PROGRAM TSCS_Bridge_Inputs	
(* Inputs from TSCS PLC to TDU PLC*)
VAR
	// Function Blocks
	BYTE_TO_BITS_10: OSCAT_BYTE_TO_BITS; // Interface for TSCS Byte 0 - Boolean inputs
	BYTE_TO_BITS_11: OSCAT_BYTE_TO_BITS; // Interface for TSCS Byte 1 - Boolean inputs
	BYTE_TO_BITS_12: OSCAT_BYTE_TO_BITS; // Interface for TSCS Byte 2 - Boolean inputs
	BYTE_TO_BITS_13: OSCAT_BYTE_TO_BITS; // Interface for TSCS Byte 3 - Boolean inputs
	BYTE_TO_BITS_14: OSCAT_BYTE_TO_BITS; // Interface for TSCS Byte 4 - Boolean inputs
	BYTE_TO_BITS_20: OSCAT_BYTE_TO_BITS; // Interface for TMS Byte 0 - Boolean inputs
	BYTE_TO_BITS_21: OSCAT_BYTE_TO_BITS; // Interface for TMS Byte 1 - Boolean inputs
	BYTE_TO_BITS_22: OSCAT_BYTE_TO_BITS; // Interface for TMS Byte 2 - Boolean inputs
	BYTE_TO_BITS_23: OSCAT_BYTE_TO_BITS; // Interface for TMS Byte 3 - Boolean inputs
	BYTE_TO_BITS_24: OSCAT_BYTE_TO_BITS; // Interface for TMS Byte 4 - Boolean inputs
	fb_Bridge_Integer_Inputs_0 : FB_Bridge_Inputs_Integer; // Interface for TSCS Integers
	fb_Bridge_Integer_Inputs_1 : FB_Bridge_Inputs_Integer; // Interface for TMS Integers
	fb_Bridge_Real_Inputs_0 : FB_Bridge_Inputs_Real; // Interface for TSCS real signals
	fb_Bridge_Real_Inputs_1 : FB_Bridge_Inputs_Real; // Interface for TMS real signals
	
	// Test Signal
	TDU_TestSignal_RB : REAL;	// Diagnostic signal readback (TDU -> TSCS ->TDU)
		
	// TSCS signals (as example)
	Lube_MainBearing_Act : BOOL; 		// Main bearing lubrication active
	TSCS_State : INT; 					// Target System Operation Mode [0=Off, 1=Normal Operation, 2=Maintenance]
	Lube_MainBearing_FlowRate : REAL; 	// Main bearing lubrication flow rate [mL/min]
END_VAR

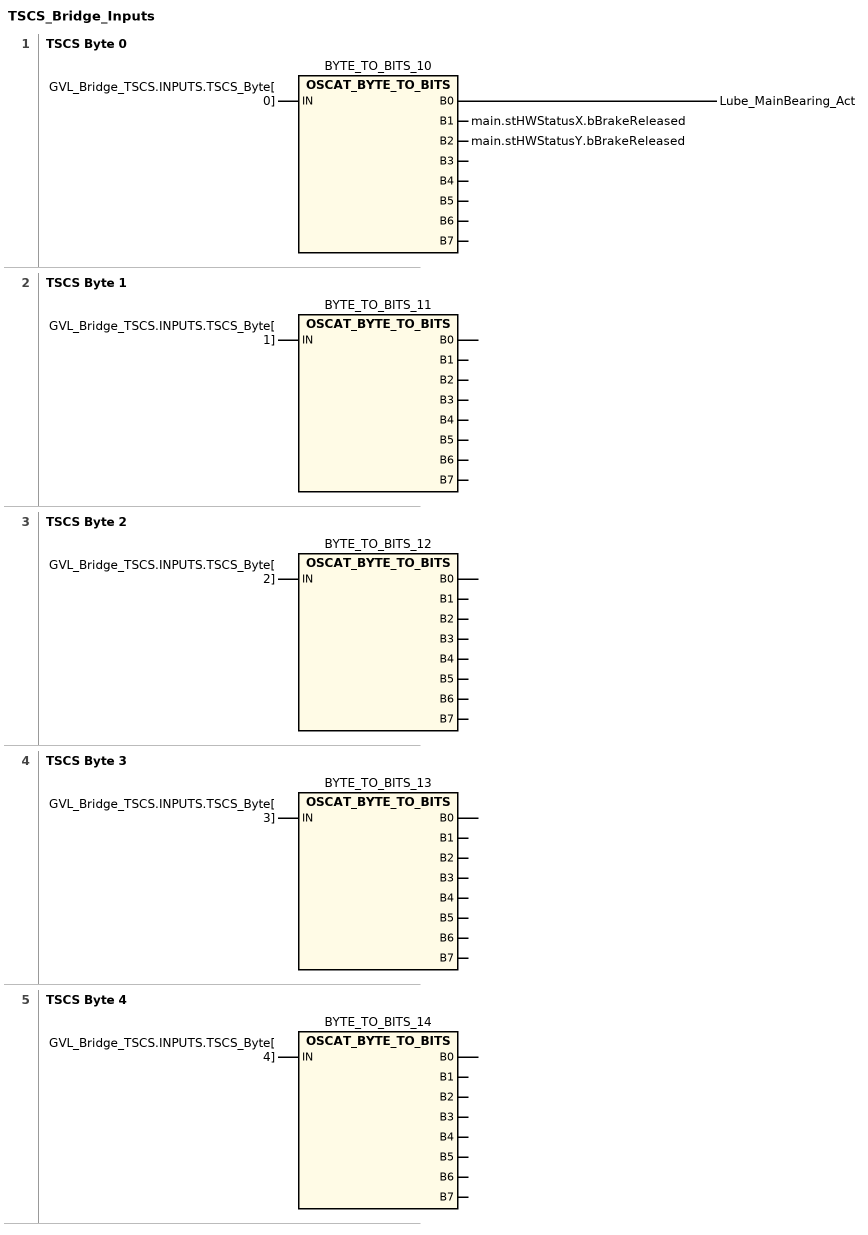
// NETWORK 1: TSCS Byte 0
BYTE_TO_BITS_10(
    IN := GVL_Bridge_TSCS.INPUTS.TSCS_Byte[0],
    B1 => main.stHWStatusX.bBrakeReleased,
    B2 => main.stHWStatusY.bBrakeReleased); // OSCAT_BYTE_TO_BITS
Lube_MainBearing_Act := BYTE_TO_BITS_10.B0;

// NETWORK 2: TSCS Byte 1
BYTE_TO_BITS_11(IN := GVL_Bridge_TSCS.INPUTS.TSCS_Byte[1]); // OSCAT_BYTE_TO_BITS

// NETWORK 3: TSCS Byte 2
BYTE_TO_BITS_12(IN := GVL_Bridge_TSCS.INPUTS.TSCS_Byte[2]); // OSCAT_BYTE_TO_BITS

// NETWORK 4: TSCS Byte 3
BYTE_TO_BITS_13(IN := GVL_Bridge_TSCS.INPUTS.TSCS_Byte[3]); // OSCAT_BYTE_TO_BITS

// NETWORK 5: TSCS Byte 4
BYTE_TO_BITS_14(IN := GVL_Bridge_TSCS.INPUTS.TSCS_Byte[4]); // OSCAT_BYTE_TO_BITS

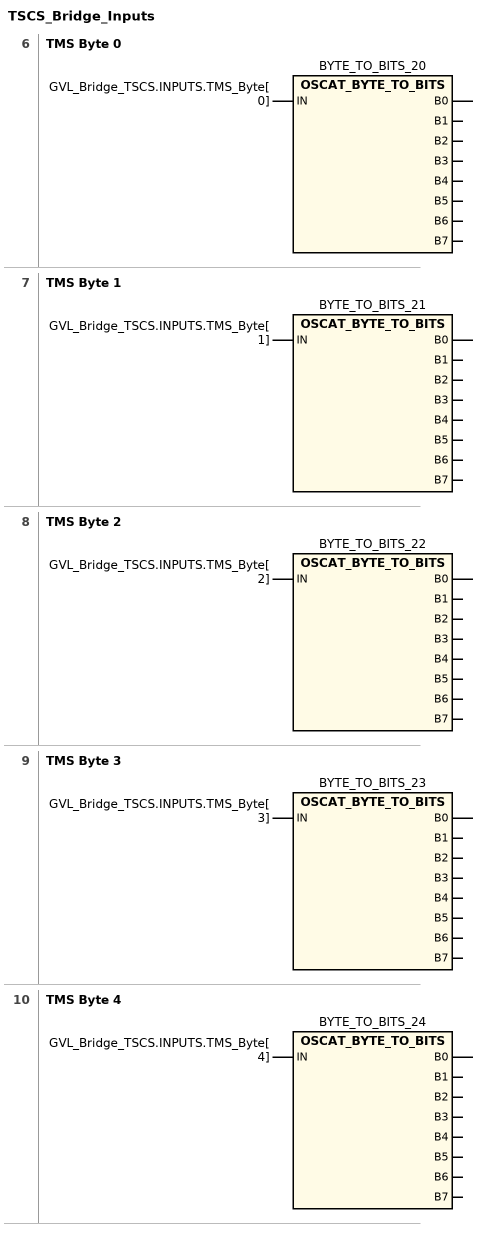
// NETWORK 6: TMS Byte 0
BYTE_TO_BITS_20(IN := GVL_Bridge_TSCS.INPUTS.TMS_Byte[0]); // OSCAT_BYTE_TO_BITS

// NETWORK 7: TMS Byte 1
BYTE_TO_BITS_21(IN := GVL_Bridge_TSCS.INPUTS.TMS_Byte[1]); // OSCAT_BYTE_TO_BITS

// NETWORK 8: TMS Byte 2
BYTE_TO_BITS_22(IN := GVL_Bridge_TSCS.INPUTS.TMS_Byte[2]); // OSCAT_BYTE_TO_BITS

// NETWORK 9: TMS Byte 3
BYTE_TO_BITS_23(IN := GVL_Bridge_TSCS.INPUTS.TMS_Byte[3]); // OSCAT_BYTE_TO_BITS

// NETWORK 10: TMS Byte 4
BYTE_TO_BITS_24(IN := GVL_Bridge_TSCS.INPUTS.TMS_Byte[4]); // OSCAT_BYTE_TO_BITS

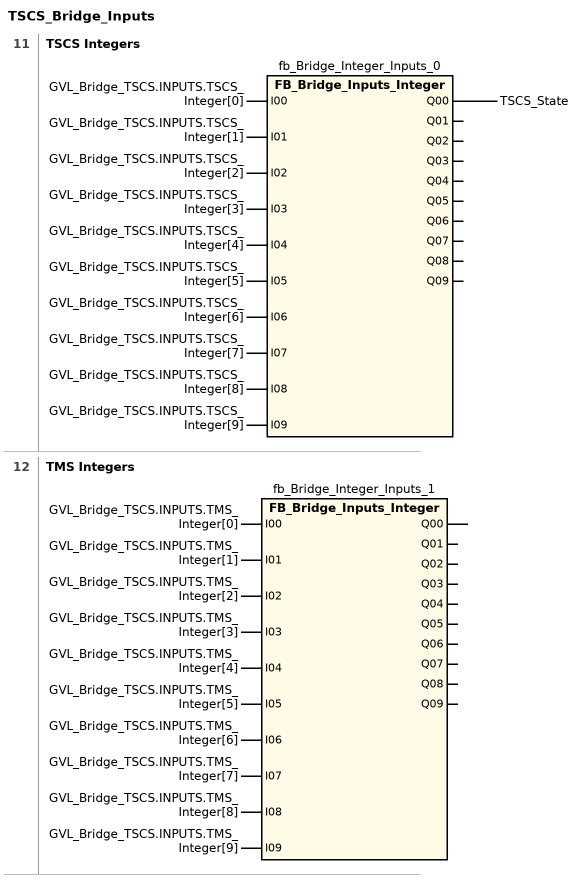
// NETWORK 11: TSCS Integers
fb_Bridge_Integer_Inputs_0(
    I00 := GVL_Bridge_TSCS.INPUTS.TSCS_Integer[0],
    I01 := GVL_Bridge_TSCS.INPUTS.TSCS_Integer[1],
    I02 := GVL_Bridge_TSCS.INPUTS.TSCS_Integer[2],
    I03 := GVL_Bridge_TSCS.INPUTS.TSCS_Integer[3],
    I04 := GVL_Bridge_TSCS.INPUTS.TSCS_Integer[4],
    I05 := GVL_Bridge_TSCS.INPUTS.TSCS_Integer[5],
    I06 := GVL_Bridge_TSCS.INPUTS.TSCS_Integer[6],
    I07 := GVL_Bridge_TSCS.INPUTS.TSCS_Integer[7],
    I08 := GVL_Bridge_TSCS.INPUTS.TSCS_Integer[8],
    I09 := GVL_Bridge_TSCS.INPUTS.TSCS_Integer[9]); // FB_Bridge_Inputs_Integer
TSCS_State := fb_Bridge_Integer_Inputs_0.Q00;

// NETWORK 12: TMS Integers
fb_Bridge_Integer_Inputs_1(
    I00 := GVL_Bridge_TSCS.INPUTS.TMS_Integer[0],
    I01 := GVL_Bridge_TSCS.INPUTS.TMS_Integer[1],
    I02 := GVL_Bridge_TSCS.INPUTS.TMS_Integer[2],
    I03 := GVL_Bridge_TSCS.INPUTS.TMS_Integer[3],
    I04 := GVL_Bridge_TSCS.INPUTS.TMS_Integer[4],
    I05 := GVL_Bridge_TSCS.INPUTS.TMS_Integer[5],
    I06 := GVL_Bridge_TSCS.INPUTS.TMS_Integer[6],
    I07 := GVL_Bridge_TSCS.INPUTS.TMS_Integer[7],
    I08 := GVL_Bridge_TSCS.INPUTS.TMS_Integer[8],
    I09 := GVL_Bridge_TSCS.INPUTS.TMS_Integer[9]); // FB_Bridge_Inputs_Integer

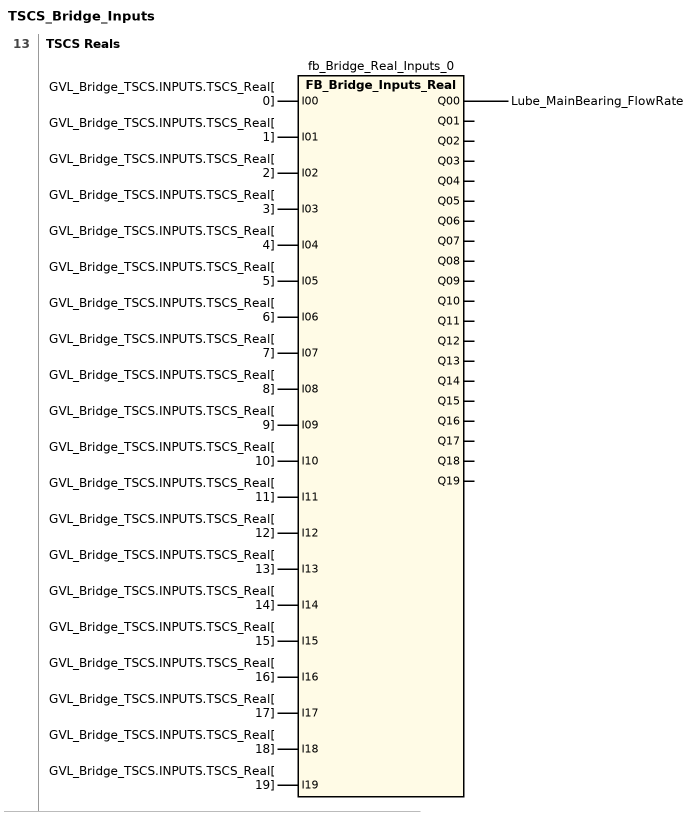
// NETWORK 13: TSCS Reals
fb_Bridge_Real_Inputs_0(
    I00 := GVL_Bridge_TSCS.INPUTS.TSCS_Real[0],
    I01 := GVL_Bridge_TSCS.INPUTS.TSCS_Real[1],
    I02 := GVL_Bridge_TSCS.INPUTS.TSCS_Real[2],
    I03 := GVL_Bridge_TSCS.INPUTS.TSCS_Real[3],
    I04 := GVL_Bridge_TSCS.INPUTS.TSCS_Real[4],
    I05 := GVL_Bridge_TSCS.INPUTS.TSCS_Real[5],
    I06 := GVL_Bridge_TSCS.INPUTS.TSCS_Real[6],
    I07 := GVL_Bridge_TSCS.INPUTS.TSCS_Real[7],
    I08 := GVL_Bridge_TSCS.INPUTS.TSCS_Real[8],
    I09 := GVL_Bridge_TSCS.INPUTS.TSCS_Real[9],
    I10 := GVL_Bridge_TSCS.INPUTS.TSCS_Real[10],
    I11 := GVL_Bridge_TSCS.INPUTS.TSCS_Real[11],
    I12 := GVL_Bridge_TSCS.INPUTS.TSCS_Real[12],
    I13 := GVL_Bridge_TSCS.INPUTS.TSCS_Real[13],
    I14 := GVL_Bridge_TSCS.INPUTS.TSCS_Real[14],
    I15 := GVL_Bridge_TSCS.INPUTS.TSCS_Real[15],
    I16 := GVL_Bridge_TSCS.INPUTS.TSCS_Real[16],
    I17 := GVL_Bridge_TSCS.INPUTS.TSCS_Real[17],
    I18 := GVL_Bridge_TSCS.INPUTS.TSCS_Real[18],
    I19 := GVL_Bridge_TSCS.INPUTS.TSCS_Real[19]); // FB_Bridge_Inputs_Real
Lube_MainBearing_FlowRate := fb_Bridge_Real_Inputs_0.Q00;

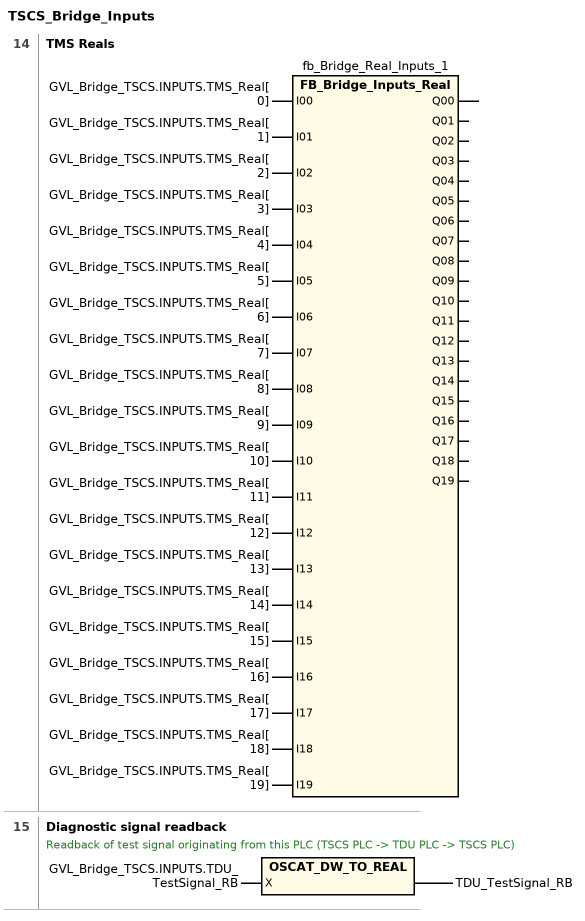
// NETWORK 14: TMS Reals
fb_Bridge_Real_Inputs_1(
    I00 := GVL_Bridge_TSCS.INPUTS.TMS_Real[0],
    I01 := GVL_Bridge_TSCS.INPUTS.TMS_Real[1],
    I02 := GVL_Bridge_TSCS.INPUTS.TMS_Real[2],
    I03 := GVL_Bridge_TSCS.INPUTS.TMS_Real[3],
    I04 := GVL_Bridge_TSCS.INPUTS.TMS_Real[4],
    I05 := GVL_Bridge_TSCS.INPUTS.TMS_Real[5],
    I06 := GVL_Bridge_TSCS.INPUTS.TMS_Real[6],
    I07 := GVL_Bridge_TSCS.INPUTS.TMS_Real[7],
    I08 := GVL_Bridge_TSCS.INPUTS.TMS_Real[8],
    I09 := GVL_Bridge_TSCS.INPUTS.TMS_Real[9],
    I10 := GVL_Bridge_TSCS.INPUTS.TMS_Real[10],
    I11 := GVL_Bridge_TSCS.INPUTS.TMS_Real[11],
    I12 := GVL_Bridge_TSCS.INPUTS.TMS_Real[12],
    I13 := GVL_Bridge_TSCS.INPUTS.TMS_Real[13],
    I14 := GVL_Bridge_TSCS.INPUTS.TMS_Real[14],
    I15 := GVL_Bridge_TSCS.INPUTS.TMS_Real[15],
    I16 := GVL_Bridge_TSCS.INPUTS.TMS_Real[16],
    I17 := GVL_Bridge_TSCS.INPUTS.TMS_Real[17],
    I18 := GVL_Bridge_TSCS.INPUTS.TMS_Real[18],
    I19 := GVL_Bridge_TSCS.INPUTS.TMS_Real[19]); // FB_Bridge_Inputs_Real

// NETWORK 15: Diagnostic signal readback
// Readback of test signal originating from this PLC (TSCS PLC -> TDU PLC -> TSCS PLC)
TDU_TestSignal_RB := OSCAT_DW_TO_REAL(X := GVL_Bridge_TSCS.INPUTS.TDU_TestSignal_RB);

END_PROGRAM

(* stored: Version 1.1.0.1, ProductVersion 3.1.4024.6
   POU TSCS_Bridge_Inputs: Id {7b91ca15-7221-418a-8914-49b2d98ef7bd}, SpecialFunc None *)
